FUNCTION_BLOCK TestComponent EXTENDS TcoCore.TcoComponent
VAR_IN_OUT
	_signal : BOOL;
END_VAR
VAR
	_signalInfo : TcoCore.TcoSignalInfo;
END_VAR

_signalInfo := THIS^.GetSignalInfo(SIZEOF(_signal), ADR(_signal));

(*~
	<docu>
		<summary>
			Restores this instance to the Ready state. Can be called explicitly or from within one of the restore mechanisms.	
		</summary>			
	</docu>	
~*)
METHOD  Restore : ITcoRestorable
END_METHOD

(*~
	<docu>
		<summary>
		    Custom service (manual, maintenance) logic.
			This method must be implemented in derived class.
		</summary>			
	</docu>	
~*)
METHOD PROTECTED  ServiceMode
END_METHOD

END_FUNCTION_BLOCK

(* stored: Version 1.1.0.1
   POU TestComponent: Id {4f004e63-6d49-073d-3db2-78e2692362d9}, SpecialFunc None
   Method Restore: Id {6ab39057-f575-055f-1d06-109a6dd5fc68}
   Method ServiceMode: Id {45b219fe-c35f-04b2-2f9b-1460cf26b4d9} *)
